PROGRAM PRG_AlarmControl
VAR CONSTANT
	sDEFAULT_NAME		: STRING := 'TwinCAT3 Event Logger';	
	sDEFAULT_FILE_PATH	: STRING := 'C:\TcEvents\';
END_VAR
VAR
	bFirstCycle			: BOOL := TRUE;
	fbAlarmControler 	: FB_AlarmControler;
	
	bInit 				: BOOL;
	bAbort				: BOOL;
END_VAR

IF bFirstCycle THEN
	bFirstCycle := FALSE;
	
	fbAlarmControler.MR_FirstCycle( sName		:= sDEFAULT_NAME,
									sFileName	:= sDEFAULT_FILE_PATH);
									
	(* Assign machine controler reference to Shell API*)
	stShell.stPlatform.ref_fbAlarmControler REF= fbAlarmControler;
	
	(* Set assignamnet done bit for visu controler *)
	stShell.stFlags.bAlarmCtrlAssignamentsDone := TRUE;
END_IF

fbAlarmControler();

END_PROGRAM

(* stored: Version 1.1.0.1, ProductVersion 3.1.4024.9
   POU PRG_AlarmControl: Id {95cce014-d1d8-4e1c-a671-e7c9ebd875d2}, SpecialFunc None *)
